(* PLC project PLC1, Beckhoff Automation GmbH TwinCAT PLC Control 3.5.13.21 *)
(* stored: creationDateTime 2023-10-06T10:55:09.0122341, modificationDateTime 2023-10-06T10:55:09.0162327 *)

PROGRAM SafeBrakeTest
  VAR
    currentIq AT %I* : DINT;
  END_VAR
  VAR
    ax1 : AXIS_REF;
    fbPower : MC_Power;
    enablePower : BOOL;
    enableTest : BOOL;
    fbBrakeTest : FB_CoEAX8000BrakeTest;
    fbBrakeCtrl : FB_CoEAX8000BrakeControl;
    fbMoveAbs : MC_MoveAbsolute;
    fbWriteDriveOpMode : MC_WriteDriveOperationMode;
    fbReadDriveOpMode : MC_ReadDriveOperationMode;
    setDriveOpMode : BOOL;
    readDriveOpMode : BOOL;
    brakeTestState : INT;
    enableMove : BOOL;
    sbtTime : TON;
    enableBrakeTest : BOOL;
  END_VAR

            fbMoveAbs(
	Axis:= ax1, 
	Execute:= , 
	Position:= , 
	Velocity:= , 
	 );

fbPower(
	Axis:= ax1, 
	Enable:= enablePower, 
	Enable_Positive:= enablePower, 
	Enable_Negative:= enablePower, 
	Override:= 100, 
	BufferMode:= , 
	Options:= , 
	Status=> , 
	Busy=> , 
	Active=> , 
	Error=> , 
	ErrorID=> );

ax1.ReadStatus();

fbBrakeTest(
	Axis:= ax1, 
	Execute:= enableBrakeTest, 
	Succeeded:= safety.SBT_Valid_PLC,
	Torque:= 0.17, 			// will vary depending on motor - value is torque that should be effective (Nm)
	VelocityLimit:= 150,	// velocity limit to prevent uncontrolled acceleration in torque mode
	Timeout := T#10S);
	
fbMoveAbs( Axis := Ax1, Execute := enableMove);
fbWriteDriveOpMode(Axis:= ax1, Execute:= setDriveOpMode);
fbReadDriveOpMode(Axis := ax1, Execute := readDriveOpMode);
sbtTime (IN := (brakeTestState=20), PT:= T#5S);

CASE brakeTestState OF
	
	0:	// is axis enabled?
		IF fbPower.Status AND enableTest THEN
			enableTest := FALSE;
			brakeTestState := 1;
		END_IF;
		
	1:	// move to safe position (0)
		fbMoveAbs.Position := 0;
		fbMoveAbs.Velocity := 250;
		enableMove := TRUE;

		IF fbMoveAbs.Busy THEN
			enableMove := FALSE;
			brakeTestState := 2;
		END_IF;		
		
	2:	// confirm in position
		IF ax1.Status.InTargetPosition THEN
			brakeTestState := 5;
		ELSIF fbMoveAbs.Error THEN
			brakeTestState := 99;
		END_IF;			
	
	5:	// engaged brake by using SBC
		safety.SBC_Enable_PLC := FALSE;
		brakeTestState := 10;
	
	10:	// switch to torque op mode
		fbWriteDriveOpMode.DriveOperationMode := DriveOperationMode_Torque;
		setDriveOpMode := TRUE;
		
		IF fbWriteDriveOpMode.Busy THEN
			setDriveOpMode := FALSE;
			brakeTestState := 11;
		ELSIF fbWriteDriveOpMode.Error THEN
			setDriveOpMode := FALSE;
			brakeTestState := 99;
		END_IF
		
	11:	// check torque op mode
		readDriveOpMode := TRUE;
		
		IF fbReadDriveOpMode.DriveOperationMode = DriveOperationMode_Torque THEN
			readDriveOpMode := FALSE;
			brakeTestState := 15;
		ELSIF fbReadDriveOpMode.Error THEN
			setDriveOpMode := FALSE;
			brakeTestState := 99;
		END_IF		
	
	15:	// start PLC brake test
		enableBrakeTest := TRUE;
		
		IF fbBrakeTest.Busy THEN
			safety.SBT_Enable_PLC := TRUE;
			brakeTestState := 20;
		ELSIF fbBrakeTest.Error THEN
			enableBrakeTest := FALSE;
			brakeTestState := 99;
		END_IF
	
	20:	// start safe brake test evaluation
	
		IF safety.SBT_Valid_PLC AND fbBrakeTest.Succeeded AND sbtTime.Q THEN
			enableBrakeTest := FALSE;
			safety.SBT_Enable_PLC := FALSE;
			safety.SBC_Enable_PLC := TRUE;
			brakeTestState := 100;
		ELSIF (safety.SBT_Error_PLC OR fbBrakeTest.Error) AND sbtTime.Q THEN
			safety.SBT_Enable_PLC := FALSE;
			brakeTestState := 99;
		END_IF
		
	100: // return back to starting operation position (500)
		readDriveOpMode := TRUE;
			
		IF fbReadDriveOpMode.DriveOperationMode = DriveOperationMode_Pos1 THEN
			fbMoveAbs.Position	:= 500;
			fbMoveAbs.Velocity	:= 250;
			enableMove			:= TRUE;
		END_IF
		
		IF fbMoveAbs.Busy THEN
			readDriveOpMode	:= FALSE;			
			enableMove		:= FALSE;
			brakeTestState := 0;
		ELSIF fbMoveAbs.Error THEN
			readDriveOpMode	:= FALSE;			
			enableMove		:= FALSE;
			brakeTestState := 99;
		END_IF
	
	
END_CASE

          
END_PROGRAM
